# EPICS autosave request: iocBoot/ioc13idd_mirror/auto_positions.req
file "CARS_4_motor_positions.req",       P=$(P)
~
